; Data for Routine_0
DECL LDAT LCPDATP1={VEL 1,ACC 100,APO_DIST 5,APO_FAC 50.0,ORI_TYP #VAR,CIRC_TYP #BASE,JERK_FAC 50.0}
DECL FDAT FP1={TOOL_NO 2,BASE_NO 10,IPO_FRAME #BASE,POINT2[] " ",TQ_STATE FALSE}
DECL E6POS XP1={X -58.570,Y 107.870,Z -38.440,A 0.000,B -17.860,C -36.410}
DECL LDAT LCPDATC2={VEL 0.1,ACC 100,APO_DIST 5,APO_FAC 50.0,ORI_TYP #VAR,CIRC_TYP #BASE,JERK_FAC 50.0}
DECL FDAT FC2={TOOL_NO 2,BASE_NO 10,IPO_FRAME #BASE,POINT2[] " ",TQ_STATE FALSE}
DECL E6POS XCAux2={X -46.970,Y 113.400,Z -38.440,A 0.000,B -14.240,C -37.780}
DECL E6POS XCDes2={X 46.970,Y 113.400,Z -38.440,A 0.000,B 14.240,C -37.780}
DECL LDAT LCPDATP3={VEL 1,ACC 100,APO_DIST 5,APO_FAC 50.0,ORI_TYP #VAR,CIRC_TYP #BASE,JERK_FAC 50.0}
DECL FDAT FP3={TOOL_NO 2,BASE_NO 10,IPO_FRAME #BASE,POINT2[] " ",TQ_STATE FALSE}
DECL E6POS XP3={X 58.570,Y 107.870,Z -38.440,A 0.000,B 17.860,C -36.410}
DECL LDAT LCPDATP4={VEL 1,ACC 100,APO_DIST 5,APO_FAC 50.0,ORI_TYP #VAR,CIRC_TYP #BASE,JERK_FAC 50.0}
DECL FDAT FP4={TOOL_NO 2,BASE_NO 10,IPO_FRAME #BASE,POINT2[] " ",TQ_STATE FALSE}
DECL E6POS XP4={X 62.100,Y 114.380,Z -43.390,A 0.000,B 12.720,C -24.560}
DECL LDAT LCPDATC5={VEL 0.1,ACC 100,APO_DIST 5,APO_FAC 50.0,ORI_TYP #VAR,CIRC_TYP #BASE,JERK_FAC 50.0}
DECL FDAT FC5={TOOL_NO 2,BASE_NO 10,IPO_FRAME #BASE,POINT2[] " ",TQ_STATE FALSE}
DECL E6POS XCAux5={X 49.810,Y 120.250,Z -43.390,A 0.000,B 10.170,C -25.660}
DECL E6POS XCDes5={X -49.810,Y 120.250,Z -43.390,A -0.000,B -10.170,C -25.660}
DECL LDAT LCPDATP6={VEL 1,ACC 100,APO_DIST 5,APO_FAC 50.0,ORI_TYP #VAR,CIRC_TYP #BASE,JERK_FAC 50.0}
DECL FDAT FP6={TOOL_NO 2,BASE_NO 10,IPO_FRAME #BASE,POINT2[] " ",TQ_STATE FALSE}
DECL E6POS XP6={X -62.100,Y 114.380,Z -43.390,A 0.000,B -12.720,C -24.560}
DECL LDAT LCPDATP7={VEL 1,ACC 100,APO_DIST 5,APO_FAC 50.0,ORI_TYP #VAR,CIRC_TYP #BASE,JERK_FAC 50.0}
DECL FDAT FP7={TOOL_NO 2,BASE_NO 10,IPO_FRAME #BASE,POINT2[] " ",TQ_STATE FALSE}
DECL E6POS XP7={X -66.070,Y 121.680,Z -46.620,A -0.000,B -7.070,C -13.210}
DECL LDAT LCPDATC8={VEL 0.1,ACC 100,APO_DIST 5,APO_FAC 50.0,ORI_TYP #VAR,CIRC_TYP #BASE,JERK_FAC 50.0}
DECL FDAT FC8={TOOL_NO 2,BASE_NO 10,IPO_FRAME #BASE,POINT2[] " ",TQ_STATE FALSE}
DECL E6POS XCAux8={X -52.990,Y 127.920,Z -46.620,A 0.000,B -5.670,C -13.860}
DECL E6POS XCDes8={X 52.990,Y 127.920,Z -46.620,A 0.000,B 5.670,C -13.860}
DECL LDAT LCPDATP9={VEL 1,ACC 100,APO_DIST 5,APO_FAC 50.0,ORI_TYP #VAR,CIRC_TYP #BASE,JERK_FAC 50.0}
DECL FDAT FP9={TOOL_NO 2,BASE_NO 10,IPO_FRAME #BASE,POINT2[] " ",TQ_STATE FALSE}
DECL E6POS XP9={X 66.070,Y 121.680,Z -46.620,A 0.000,B 7.070,C -13.210}
DECL LDAT LCPDATP10={VEL 1,ACC 100,APO_DIST 5,APO_FAC 50.0,ORI_TYP #VAR,CIRC_TYP #BASE,JERK_FAC 50.0}
DECL FDAT FP10={TOOL_NO 2,BASE_NO 10,IPO_FRAME #BASE,POINT2[] " ",TQ_STATE FALSE}
DECL E6POS XP10={X 70.270,Y 129.420,Z -47.960,A 0.000,B 1.160,C -2.140}
DECL LDAT LCPDATC11={VEL 0.1,ACC 100,APO_DIST 5,APO_FAC 50.0,ORI_TYP #VAR,CIRC_TYP #BASE,JERK_FAC 50.0}
DECL FDAT FC11={TOOL_NO 2,BASE_NO 10,IPO_FRAME #BASE,POINT2[] " ",TQ_STATE FALSE}
DECL E6POS XCAux11={X 56.360,Y 136.060,Z -47.960,A 0.000,B 0.930,C -2.250}
DECL E6POS XCDes11={X -56.360,Y 136.060,Z -47.960,A 0.000,B -0.930,C -2.250}
DECL LDAT LCPDATP12={VEL 1,ACC 100,APO_DIST 5,APO_FAC 50.0,ORI_TYP #VAR,CIRC_TYP #BASE,JERK_FAC 50.0}
DECL FDAT FP12={TOOL_NO 2,BASE_NO 10,IPO_FRAME #BASE,POINT2[] " ",TQ_STATE FALSE}
DECL E6POS XP12={X -70.270,Y 129.420,Z -47.960,A 0.000,B -1.160,C -2.140}
DECL LDAT LCPDATP13={VEL 1,ACC 100,APO_DIST 5,APO_FAC 50.0,ORI_TYP #VAR,CIRC_TYP #BASE,JERK_FAC 50.0}
DECL FDAT FP13={TOOL_NO 2,BASE_NO 10,IPO_FRAME #BASE,POINT2[] " ",TQ_STATE FALSE}
DECL E6POS XP13={X -70.330,Y 129.530,Z -48.000,A 0.000,B 0.000,C -0.000}
DECL LDAT LCPDATC14={VEL 0.1,ACC 100,APO_DIST 5,APO_FAC 50.0,ORI_TYP #VAR,CIRC_TYP #BASE,JERK_FAC 50.0}
DECL FDAT FC14={TOOL_NO 2,BASE_NO 10,IPO_FRAME #BASE,POINT2[] " ",TQ_STATE FALSE}
DECL E6POS XCAux14={X -56.400,Y 136.170,Z -48.000,A 0.000,B 0.000,C -0.000}
DECL E6POS XCDes14={X 56.400,Y 136.170,Z -48.000,A 0.000,B 0.000,C -0.000}
DECL LDAT LCPDATP15={VEL 1,ACC 100,APO_DIST 5,APO_FAC 50.0,ORI_TYP #VAR,CIRC_TYP #BASE,JERK_FAC 50.0}
DECL FDAT FP15={TOOL_NO 2,BASE_NO 10,IPO_FRAME #BASE,POINT2[] " ",TQ_STATE FALSE}
DECL E6POS XP15={X 70.330,Y 129.530,Z -48.000,A 0.000,B 0.000,C -0.000}
DECL LDAT LCPDATP16={VEL 1,ACC 100,APO_DIST 5,APO_FAC 50.0,ORI_TYP #VAR,CIRC_TYP #BASE,JERK_FAC 50.0}
DECL FDAT FP16={TOOL_NO 2,BASE_NO 10,IPO_FRAME #BASE,POINT2[] " ",TQ_STATE FALSE}
DECL E6POS XP16={X 69.370,Y 127.770,Z -48.000,A 0.000,B 0.000,C -0.000}
DECL LDAT LCPDATC17={VEL 0.1,ACC 100,APO_DIST 5,APO_FAC 50.0,ORI_TYP #VAR,CIRC_TYP #BASE,JERK_FAC 50.0}
DECL FDAT FC17={TOOL_NO 2,BASE_NO 10,IPO_FRAME #BASE,POINT2[] " ",TQ_STATE FALSE}
DECL E6POS XCAux17={X 55.640,Y 134.320,Z -48.000,A 0.000,B 0.000,C -0.000}
DECL E6POS XCDes17={X -55.640,Y 134.320,Z -48.000,A 0.000,B 0.000,C -0.000}
DECL LDAT LCPDATP18={VEL 1,ACC 100,APO_DIST 5,APO_FAC 50.0,ORI_TYP #VAR,CIRC_TYP #BASE,JERK_FAC 50.0}
DECL FDAT FP18={TOOL_NO 2,BASE_NO 10,IPO_FRAME #BASE,POINT2[] " ",TQ_STATE FALSE}
DECL E6POS XP18={X -69.370,Y 127.770,Z -48.000,A 0.000,B 0.000,C -0.000}
DECL LDAT LCPDATP19={VEL 1,ACC 100,APO_DIST 5,APO_FAC 50.0,ORI_TYP #VAR,CIRC_TYP #BASE,JERK_FAC 50.0}
DECL FDAT FP19={TOOL_NO 2,BASE_NO 10,IPO_FRAME #BASE,POINT2[] " ",TQ_STATE FALSE}
DECL E6POS XP19={X -68.420,Y 126.010,Z -48.000,A 0.000,B 0.000,C -0.000}
DECL LDAT LCPDATC20={VEL 0.1,ACC 100,APO_DIST 5,APO_FAC 50.0,ORI_TYP #VAR,CIRC_TYP #BASE,JERK_FAC 50.0}
DECL FDAT FC20={TOOL_NO 2,BASE_NO 10,IPO_FRAME #BASE,POINT2[] " ",TQ_STATE FALSE}
DECL E6POS XCAux20={X -54.870,Y 132.470,Z -48.000,A 0.000,B 0.000,C -0.000}
DECL E6POS XCDes20={X 54.870,Y 132.470,Z -48.000,A 0.000,B 0.000,C -0.000}
DECL LDAT LCPDATP21={VEL 1,ACC 100,APO_DIST 5,APO_FAC 50.0,ORI_TYP #VAR,CIRC_TYP #BASE,JERK_FAC 50.0}
DECL FDAT FP21={TOOL_NO 2,BASE_NO 10,IPO_FRAME #BASE,POINT2[] " ",TQ_STATE FALSE}
DECL E6POS XP21={X 68.420,Y 126.010,Z -48.000,A 0.000,B 0.000,C -0.000}
DECL LDAT LCPDATP22={VEL 1,ACC 100,APO_DIST 5,APO_FAC 50.0,ORI_TYP #VAR,CIRC_TYP #BASE,JERK_FAC 50.0}
DECL FDAT FP22={TOOL_NO 2,BASE_NO 10,IPO_FRAME #BASE,POINT2[] " ",TQ_STATE FALSE}
DECL E6POS XP22={X 67.460,Y 124.250,Z -48.000,A 0.000,B 0.000,C -0.000}
DECL LDAT LCPDATC23={VEL 0.1,ACC 100,APO_DIST 5,APO_FAC 50.0,ORI_TYP #VAR,CIRC_TYP #BASE,JERK_FAC 50.0}
DECL FDAT FC23={TOOL_NO 2,BASE_NO 10,IPO_FRAME #BASE,POINT2[] " ",TQ_STATE FALSE}
DECL E6POS XCAux23={X 54.110,Y 130.630,Z -48.000,A 0.000,B 0.000,C -0.000}
DECL E6POS XCDes23={X -54.110,Y 130.630,Z -48.000,A 0.000,B 0.000,C -0.000}
DECL LDAT LCPDATP24={VEL 1,ACC 100,APO_DIST 5,APO_FAC 50.0,ORI_TYP #VAR,CIRC_TYP #BASE,JERK_FAC 50.0}
DECL FDAT FP24={TOOL_NO 2,BASE_NO 10,IPO_FRAME #BASE,POINT2[] " ",TQ_STATE FALSE}
DECL E6POS XP24={X -67.460,Y 124.250,Z -48.000,A 0.000,B 0.000,C -0.000}
DECL LDAT LCPDATP25={VEL 1,ACC 100,APO_DIST 5,APO_FAC 50.0,ORI_TYP #VAR,CIRC_TYP #BASE,JERK_FAC 50.0}
DECL FDAT FP25={TOOL_NO 2,BASE_NO 10,IPO_FRAME #BASE,POINT2[] " ",TQ_STATE FALSE}
DECL E6POS XP25={X -70.710,Y 130.240,Z -47.360,A 0.000,B 4.820,C 8.940}
DECL LDAT LCPDATC26={VEL 0.1,ACC 100,APO_DIST 5,APO_FAC 50.0,ORI_TYP #VAR,CIRC_TYP #BASE,JERK_FAC 50.0}
DECL FDAT FC26={TOOL_NO 2,BASE_NO 10,IPO_FRAME #BASE,POINT2[] " ",TQ_STATE FALSE}
DECL E6POS XCAux26={X -56.710,Y 136.910,Z -47.360,A 0.000,B 3.870,C 9.390}
DECL E6POS XCDes26={X 56.710,Y 136.910,Z -47.360,A 0.000,B -3.870,C 9.390}
DECL LDAT LCPDATP27={VEL 1,ACC 100,APO_DIST 5,APO_FAC 50.0,ORI_TYP #VAR,CIRC_TYP #BASE,JERK_FAC 50.0}
DECL FDAT FP27={TOOL_NO 2,BASE_NO 10,IPO_FRAME #BASE,POINT2[] " ",TQ_STATE FALSE}
DECL E6POS XP27={X 70.710,Y 130.240,Z -47.360,A -0.000,B -4.820,C 8.940}
DECL LDAT LCPDATP28={VEL 1,ACC 100,APO_DIST 5,APO_FAC 50.0,ORI_TYP #VAR,CIRC_TYP #BASE,JERK_FAC 50.0}
DECL FDAT FP28={TOOL_NO 2,BASE_NO 10,IPO_FRAME #BASE,POINT2[] " ",TQ_STATE FALSE}
DECL E6POS XP28={X 74.790,Y 137.750,Z -44.840,A -0.000,B -10.600,C 20.160}
DECL LDAT LCPDATC29={VEL 0.1,ACC 100,APO_DIST 5,APO_FAC 50.0,ORI_TYP #VAR,CIRC_TYP #BASE,JERK_FAC 50.0}
DECL FDAT FC29={TOOL_NO 2,BASE_NO 10,IPO_FRAME #BASE,POINT2[] " ",TQ_STATE FALSE}
DECL E6POS XCAux29={X 59.980,Y 144.810,Z -44.840,A -0.000,B -8.480,C 21.100}
DECL E6POS XCDes29={X -59.980,Y 144.810,Z -44.840,A -0.000,B 8.480,C 21.100}
DECL LDAT LCPDATP30={VEL 1,ACC 100,APO_DIST 5,APO_FAC 50.0,ORI_TYP #VAR,CIRC_TYP #BASE,JERK_FAC 50.0}
DECL FDAT FP30={TOOL_NO 2,BASE_NO 10,IPO_FRAME #BASE,POINT2[] " ",TQ_STATE FALSE}
DECL E6POS XP30={X -74.790,Y 137.750,Z -44.840,A 0.000,B 10.600,C 20.160}
DECL LDAT LCPDATP31={VEL 1,ACC 100,APO_DIST 5,APO_FAC 50.0,ORI_TYP #VAR,CIRC_TYP #BASE,JERK_FAC 50.0}
DECL FDAT FP31={TOOL_NO 2,BASE_NO 10,IPO_FRAME #BASE,POINT2[] " ",TQ_STATE FALSE}
DECL E6POS XP31={X -78.510,Y 144.600,Z -40.530,A 0.000,B 15.960,C 31.790}
DECL LDAT LCPDATC32={VEL 0.1,ACC 100,APO_DIST 5,APO_FAC 50.0,ORI_TYP #VAR,CIRC_TYP #BASE,JERK_FAC 50.0}
DECL FDAT FC32={TOOL_NO 2,BASE_NO 10,IPO_FRAME #BASE,POINT2[] " ",TQ_STATE FALSE}
DECL E6POS XCAux32={X -62.970,Y 152.020,Z -40.530,A 0.000,B 12.740,C 33.080}
DECL E6POS XCDes32={X 62.970,Y 152.020,Z -40.530,A 0.000,B -12.740,C 33.080}
DECL LDAT LCPDATP33={VEL 1,ACC 100,APO_DIST 5,APO_FAC 50.0,ORI_TYP #VAR,CIRC_TYP #BASE,JERK_FAC 50.0}
DECL FDAT FP33={TOOL_NO 2,BASE_NO 10,IPO_FRAME #BASE,POINT2[] " ",TQ_STATE FALSE}
DECL E6POS XP33={X 78.510,Y 144.600,Z -40.530,A 0.000,B -15.960,C 31.790}
DECL LDAT LCPDATP34={VEL 1,ACC 100,APO_DIST 5,APO_FAC 50.0,ORI_TYP #VAR,CIRC_TYP #BASE,JERK_FAC 50.0}
DECL FDAT FP34={TOOL_NO 2,BASE_NO 10,IPO_FRAME #BASE,POINT2[] " ",TQ_STATE FALSE}
DECL E6POS XP34={X 81.700,Y 150.470,Z -34.640,A 0.000,B -20.670,C 44.020}
DECL LDAT LCPDATC35={VEL 0.1,ACC 100,APO_DIST 5,APO_FAC 50.0,ORI_TYP #VAR,CIRC_TYP #BASE,JERK_FAC 50.0}
DECL FDAT FC35={TOOL_NO 2,BASE_NO 10,IPO_FRAME #BASE,POINT2[] " ",TQ_STATE FALSE}
DECL E6POS XCAux35={X 65.520,Y 158.190,Z -34.640,A 0.000,B -16.450,C 45.450}
DECL E6POS XCDes35={X -65.520,Y 158.190,Z -34.640,A 0.000,B 16.450,C 45.450}
DECL LDAT LCPDATP36={VEL 1,ACC 100,APO_DIST 5,APO_FAC 50.0,ORI_TYP #VAR,CIRC_TYP #BASE,JERK_FAC 50.0}
DECL FDAT FP36={TOOL_NO 2,BASE_NO 10,IPO_FRAME #BASE,POINT2[] " ",TQ_STATE FALSE}
DECL E6POS XP36={X -81.700,Y 150.470,Z -34.640,A 0.000,B 20.670,C 44.020}
DECL LDAT LCPDATP37={VEL 1,ACC 100,APO_DIST 5,APO_FAC 50.0,ORI_TYP #VAR,CIRC_TYP #BASE,JERK_FAC 50.0}
DECL FDAT FP37={TOOL_NO 2,BASE_NO 10,IPO_FRAME #BASE,POINT2[] " ",TQ_STATE FALSE}
DECL E6POS XP37={X -79.930,Y 147.210,Z -38.750,A -0.000,B 17.860,C 36.410}
DECL LDAT LCPDATC38={VEL 0.1,ACC 100,APO_DIST 5,APO_FAC 50.0,ORI_TYP #VAR,CIRC_TYP #BASE,JERK_FAC 50.0}
DECL FDAT FC38={TOOL_NO 2,BASE_NO 10,IPO_FRAME #BASE,POINT2[] " ",TQ_STATE FALSE}
DECL E6POS XCAux38={X -64.110,Y 154.760,Z -38.750,A -0.000,B 14.240,C 37.780}
DECL E6POS XCDes38={X 64.110,Y 154.760,Z -38.750,A 0.000,B -14.240,C 37.780}
DECL LDAT LCPDATP39={VEL 1,ACC 100,APO_DIST 5,APO_FAC 50.0,ORI_TYP #VAR,CIRC_TYP #BASE,JERK_FAC 50.0}
DECL FDAT FP39={TOOL_NO 2,BASE_NO 10,IPO_FRAME #BASE,POINT2[] " ",TQ_STATE FALSE}
DECL E6POS XP39={X 79.930,Y 147.210,Z -38.750,A -0.000,B -17.860,C 36.410}
DECL LDAT LCPDATP40={VEL 1,ACC 100,APO_DIST 5,APO_FAC 50.0,ORI_TYP #VAR,CIRC_TYP #BASE,JERK_FAC 50.0}
DECL FDAT FP40={TOOL_NO 2,BASE_NO 10,IPO_FRAME #BASE,POINT2[] " ",TQ_STATE FALSE}
DECL E6POS XP40={X 76.190,Y 140.320,Z -43.940,A -0.000,B -12.470,C 24.030}
DECL LDAT LCPDATC41={VEL 0.1,ACC 100,APO_DIST 5,APO_FAC 50.0,ORI_TYP #VAR,CIRC_TYP #BASE,JERK_FAC 50.0}
DECL FDAT FC41={TOOL_NO 2,BASE_NO 10,IPO_FRAME #BASE,POINT2[] " ",TQ_STATE FALSE}
DECL E6POS XCAux41={X 61.100,Y 147.510,Z -43.940,A -0.000,B -9.970,C 25.120}
DECL E6POS XCDes41={X -61.100,Y 147.510,Z -43.940,A 0.000,B 9.970,C 25.120}
DECL LDAT LCPDATP42={VEL 1,ACC 100,APO_DIST 5,APO_FAC 50.0,ORI_TYP #VAR,CIRC_TYP #BASE,JERK_FAC 50.0}
DECL FDAT FP42={TOOL_NO 2,BASE_NO 10,IPO_FRAME #BASE,POINT2[] " ",TQ_STATE FALSE}
DECL E6POS XP42={X -76.190,Y 140.320,Z -43.940,A 0.000,B 12.470,C 24.030}
DECL LDAT LCPDATP43={VEL 1,ACC 100,APO_DIST 5,APO_FAC 50.0,ORI_TYP #VAR,CIRC_TYP #BASE,JERK_FAC 50.0}
DECL FDAT FP43={TOOL_NO 2,BASE_NO 10,IPO_FRAME #BASE,POINT2[] " ",TQ_STATE FALSE}
DECL E6POS XP43={X -71.980,Y 132.570,Z -47.210,A 0.000,B 6.540,C 12.190}
DECL LDAT LCPDATC44={VEL 0.1,ACC 100,APO_DIST 5,APO_FAC 50.0,ORI_TYP #VAR,CIRC_TYP #BASE,JERK_FAC 50.0}
DECL FDAT FC44={TOOL_NO 2,BASE_NO 10,IPO_FRAME #BASE,POINT2[] " ",TQ_STATE FALSE}
DECL E6POS XCAux44={X -57.730,Y 139.360,Z -47.210,A 0.000,B 5.240,C 12.790}
DECL E6POS XCDes44={X 57.730,Y 139.360,Z -47.210,A 0.000,B -5.240,C 12.790}
DECL LDAT LCPDATP45={VEL 1,ACC 100,APO_DIST 5,APO_FAC 50.0,ORI_TYP #VAR,CIRC_TYP #BASE,JERK_FAC 50.0}
DECL FDAT FP45={TOOL_NO 2,BASE_NO 10,IPO_FRAME #BASE,POINT2[] " ",TQ_STATE FALSE}
DECL E6POS XP45={X 71.980,Y 132.570,Z -47.210,A 0.000,B -6.540,C 12.190}
DECL LDAT LCPDATP46={VEL 1,ACC 100,APO_DIST 5,APO_FAC 50.0,ORI_TYP #VAR,CIRC_TYP #BASE,JERK_FAC 50.0}
DECL FDAT FP46={TOOL_NO 2,BASE_NO 10,IPO_FRAME #BASE,POINT2[] " ",TQ_STATE FALSE}
DECL E6POS XP46={X 67.520,Y 124.360,Z -48.400,A 0.000,B -0.340,C 0.630}
DECL LDAT LCPDATC47={VEL 0.1,ACC 100,APO_DIST 5,APO_FAC 50.0,ORI_TYP #VAR,CIRC_TYP #BASE,JERK_FAC 50.0}
DECL FDAT FC47={TOOL_NO 2,BASE_NO 10,IPO_FRAME #BASE,POINT2[] " ",TQ_STATE FALSE}
DECL E6POS XCAux47={X 54.160,Y 130.740,Z -48.400,A -0.000,B -0.270,C 0.660}
DECL E6POS XCDes47={X -54.160,Y 130.740,Z -48.400,A 0.000,B 0.270,C 0.660}
DECL LDAT LCPDATP48={VEL 1,ACC 100,APO_DIST 5,APO_FAC 50.0,ORI_TYP #VAR,CIRC_TYP #BASE,JERK_FAC 50.0}
DECL FDAT FP48={TOOL_NO 2,BASE_NO 10,IPO_FRAME #BASE,POINT2[] " ",TQ_STATE FALSE}
DECL E6POS XP48={X -67.520,Y 124.360,Z -48.400,A 0.000,B 0.340,C 0.630}
DECL LDAT LCPDATP49={VEL 1,ACC 100,APO_DIST 5,APO_FAC 50.0,ORI_TYP #VAR,CIRC_TYP #BASE,JERK_FAC 50.0}
DECL FDAT FP49={TOOL_NO 2,BASE_NO 10,IPO_FRAME #BASE,POINT2[] " ",TQ_STATE FALSE}
DECL E6POS XP49={X -68.180,Y 125.580,Z -48.400,A 0.000,B 0.000,C -0.000}
DECL LDAT LCPDATC50={VEL 0.1,ACC 100,APO_DIST 5,APO_FAC 50.0,ORI_TYP #VAR,CIRC_TYP #BASE,JERK_FAC 50.0}
DECL FDAT FC50={TOOL_NO 2,BASE_NO 10,IPO_FRAME #BASE,POINT2[] " ",TQ_STATE FALSE}
DECL E6POS XCAux50={X -54.680,Y 132.010,Z -48.400,A 0.000,B 0.000,C -0.000}
DECL E6POS XCDes50={X 54.680,Y 132.010,Z -48.400,A 0.000,B 0.000,C -0.000}
DECL LDAT LCPDATP51={VEL 1,ACC 100,APO_DIST 5,APO_FAC 50.0,ORI_TYP #VAR,CIRC_TYP #BASE,JERK_FAC 50.0}
DECL FDAT FP51={TOOL_NO 2,BASE_NO 10,IPO_FRAME #BASE,POINT2[] " ",TQ_STATE FALSE}
DECL E6POS XP51={X 68.180,Y 125.580,Z -48.400,A 0.000,B 0.000,C -0.000}
DECL LDAT LCPDATP52={VEL 1,ACC 100,APO_DIST 5,APO_FAC 50.0,ORI_TYP #VAR,CIRC_TYP #BASE,JERK_FAC 50.0}
DECL FDAT FP52={TOOL_NO 2,BASE_NO 10,IPO_FRAME #BASE,POINT2[] " ",TQ_STATE FALSE}
DECL E6POS XP52={X 69.140,Y 127.330,Z -48.400,A 0.000,B 0.000,C -0.000}
DECL LDAT LCPDATC53={VEL 0.1,ACC 100,APO_DIST 5,APO_FAC 50.0,ORI_TYP #VAR,CIRC_TYP #BASE,JERK_FAC 50.0}
DECL FDAT FC53={TOOL_NO 2,BASE_NO 10,IPO_FRAME #BASE,POINT2[] " ",TQ_STATE FALSE}
DECL E6POS XCAux53={X 55.450,Y 133.860,Z -48.400,A 0.000,B 0.000,C -0.000}
DECL E6POS XCDes53={X -55.450,Y 133.860,Z -48.400,A 0.000,B 0.000,C -0.000}
DECL LDAT LCPDATP54={VEL 1,ACC 100,APO_DIST 5,APO_FAC 50.0,ORI_TYP #VAR,CIRC_TYP #BASE,JERK_FAC 50.0}
DECL FDAT FP54={TOOL_NO 2,BASE_NO 10,IPO_FRAME #BASE,POINT2[] " ",TQ_STATE FALSE}
DECL E6POS XP54={X -69.140,Y 127.330,Z -48.400,A 0.000,B 0.000,C -0.000}
DECL LDAT LCPDATP55={VEL 1,ACC 100,APO_DIST 5,APO_FAC 50.0,ORI_TYP #VAR,CIRC_TYP #BASE,JERK_FAC 50.0}
DECL FDAT FP55={TOOL_NO 2,BASE_NO 10,IPO_FRAME #BASE,POINT2[] " ",TQ_STATE FALSE}
DECL E6POS XP55={X -70.090,Y 129.090,Z -48.400,A 0.000,B 0.000,C -0.000}
DECL LDAT LCPDATC56={VEL 0.1,ACC 100,APO_DIST 5,APO_FAC 50.0,ORI_TYP #VAR,CIRC_TYP #BASE,JERK_FAC 50.0}
DECL FDAT FC56={TOOL_NO 2,BASE_NO 10,IPO_FRAME #BASE,POINT2[] " ",TQ_STATE FALSE}
DECL E6POS XCAux56={X -56.210,Y 135.710,Z -48.400,A 0.000,B 0.000,C -0.000}
DECL E6POS XCDes56={X 56.210,Y 135.710,Z -48.400,A 0.000,B 0.000,C -0.000}
DECL LDAT LCPDATP57={VEL 1,ACC 100,APO_DIST 5,APO_FAC 50.0,ORI_TYP #VAR,CIRC_TYP #BASE,JERK_FAC 50.0}
DECL FDAT FP57={TOOL_NO 2,BASE_NO 10,IPO_FRAME #BASE,POINT2[] " ",TQ_STATE FALSE}
DECL E6POS XP57={X 70.090,Y 129.090,Z -48.400,A 0.000,B 0.000,C -0.000}
DECL LDAT LCPDATP58={VEL 1,ACC 100,APO_DIST 5,APO_FAC 50.0,ORI_TYP #VAR,CIRC_TYP #BASE,JERK_FAC 50.0}
DECL FDAT FP58={TOOL_NO 2,BASE_NO 10,IPO_FRAME #BASE,POINT2[] " ",TQ_STATE FALSE}
DECL E6POS XP58={X 71.040,Y 130.850,Z -48.400,A 0.000,B 0.000,C -0.000}
DECL LDAT LCPDATC59={VEL 0.1,ACC 100,APO_DIST 5,APO_FAC 50.0,ORI_TYP #VAR,CIRC_TYP #BASE,JERK_FAC 50.0}
DECL FDAT FC59={TOOL_NO 2,BASE_NO 10,IPO_FRAME #BASE,POINT2[] " ",TQ_STATE FALSE}
DECL E6POS XCAux59={X 56.980,Y 137.560,Z -48.400,A 0.000,B 0.000,C -0.000}
DECL E6POS XCDes59={X -56.980,Y 137.560,Z -48.400,A 0.000,B 0.000,C -0.000}
DECL LDAT LCPDATP60={VEL 1,ACC 100,APO_DIST 5,APO_FAC 50.0,ORI_TYP #VAR,CIRC_TYP #BASE,JERK_FAC 50.0}
DECL FDAT FP60={TOOL_NO 2,BASE_NO 10,IPO_FRAME #BASE,POINT2[] " ",TQ_STATE FALSE}
DECL E6POS XP60={X -71.040,Y 130.850,Z -48.400,A 0.000,B 0.000,C -0.000}
DECL LDAT LCPDATP61={VEL 1,ACC 100,APO_DIST 5,APO_FAC 50.0,ORI_TYP #VAR,CIRC_TYP #BASE,JERK_FAC 50.0}
DECL FDAT FP61={TOOL_NO 2,BASE_NO 10,IPO_FRAME #BASE,POINT2[] " ",TQ_STATE FALSE}
DECL E6POS XP61={X -66.840,Y 123.110,Z -47.430,A 0.000,B -5.920,C -11.010}
DECL LDAT LCPDATC62={VEL 0.1,ACC 100,APO_DIST 5,APO_FAC 50.0,ORI_TYP #VAR,CIRC_TYP #BASE,JERK_FAC 50.0}
DECL FDAT FC62={TOOL_NO 2,BASE_NO 10,IPO_FRAME #BASE,POINT2[] " ",TQ_STATE FALSE}
DECL E6POS XCAux62={X -53.610,Y 129.420,Z -47.430,A 0.000,B -4.740,C -11.560}
DECL E6POS XCDes62={X 53.610,Y 129.420,Z -47.430,A 0.000,B 4.740,C -11.560}
DECL LDAT LCPDATP63={VEL 1,ACC 100,APO_DIST 5,APO_FAC 50.0,ORI_TYP #VAR,CIRC_TYP #BASE,JERK_FAC 50.0}
DECL FDAT FP63={TOOL_NO 2,BASE_NO 10,IPO_FRAME #BASE,POINT2[] " ",TQ_STATE FALSE}
DECL E6POS XP63={X 66.840,Y 123.110,Z -47.430,A 0.000,B 5.920,C -11.010}
DECL LDAT LCPDATP64={VEL 1,ACC 100,APO_DIST 5,APO_FAC 50.0,ORI_TYP #VAR,CIRC_TYP #BASE,JERK_FAC 50.0}
DECL FDAT FP64={TOOL_NO 2,BASE_NO 10,IPO_FRAME #BASE,POINT2[] " ",TQ_STATE FALSE}
DECL E6POS XP64={X 62.600,Y 115.290,Z -44.360,A 0.000,B 11.890,C -22.810}
DECL LDAT LCPDATC65={VEL 0.1,ACC 100,APO_DIST 5,APO_FAC 50.0,ORI_TYP #VAR,CIRC_TYP #BASE,JERK_FAC 50.0}
DECL FDAT FC65={TOOL_NO 2,BASE_NO 10,IPO_FRAME #BASE,POINT2[] " ",TQ_STATE FALSE}
DECL E6POS XCAux65={X 50.210,Y 121.210,Z -44.360,A 0.000,B 9.510,C -23.850}
DECL E6POS XCDes65={X -50.210,Y 121.210,Z -44.360,A 0.000,B -9.510,C -23.850}
DECL LDAT LCPDATP66={VEL 1,ACC 100,APO_DIST 5,APO_FAC 50.0,ORI_TYP #VAR,CIRC_TYP #BASE,JERK_FAC 50.0}
DECL FDAT FP66={TOOL_NO 2,BASE_NO 10,IPO_FRAME #BASE,POINT2[] " ",TQ_STATE FALSE}
DECL E6POS XP66={X -62.600,Y 115.290,Z -44.360,A 0.000,B -11.890,C -22.810}
DECL LDAT LCPDATP67={VEL 1,ACC 100,APO_DIST 5,APO_FAC 50.0,ORI_TYP #VAR,CIRC_TYP #BASE,JERK_FAC 50.0}
DECL FDAT FP67={TOOL_NO 2,BASE_NO 10,IPO_FRAME #BASE,POINT2[] " ",TQ_STATE FALSE}
DECL E6POS XP67={X -58.800,Y 108.290,Z -39.360,A -0.000,B -17.350,C -35.120}
DECL LDAT LCPDATC68={VEL 0.1,ACC 100,APO_DIST 5,APO_FAC 50.0,ORI_TYP #VAR,CIRC_TYP #BASE,JERK_FAC 50.0}
DECL FDAT FC68={TOOL_NO 2,BASE_NO 10,IPO_FRAME #BASE,POINT2[] " ",TQ_STATE FALSE}
DECL E6POS XCAux68={X -47.160,Y 113.850,Z -39.360,A 0.000,B -13.830,C -36.480}
DECL E6POS XCDes68={X 47.160,Y 113.850,Z -39.360,A 0.000,B 13.830,C -36.480}
DECL LDAT LCPDATP69={VEL 1,ACC 100,APO_DIST 5,APO_FAC 50.0,ORI_TYP #VAR,CIRC_TYP #BASE,JERK_FAC 50.0}
DECL FDAT FP69={TOOL_NO 2,BASE_NO 10,IPO_FRAME #BASE,POINT2[] " ",TQ_STATE FALSE}
DECL E6POS XP69={X 58.800,Y 108.290,Z -39.360,A 0.000,B 17.350,C -35.120}
DECL LDAT LCPDATP70={VEL 1,ACC 100,APO_DIST 5,APO_FAC 50.0,ORI_TYP #VAR,CIRC_TYP #BASE,JERK_FAC 50.0}
DECL FDAT FP70={TOOL_NO 2,BASE_NO 10,IPO_FRAME #BASE,POINT2[] " ",TQ_STATE FALSE}
DECL E6POS XP70={X 58.320,Y 107.420,Z -39.060,A -0.000,B 17.860,C -36.410}
DECL LDAT LCPDATC71={VEL 0.1,ACC 100,APO_DIST 5,APO_FAC 50.0,ORI_TYP #VAR,CIRC_TYP #BASE,JERK_FAC 50.0}
DECL FDAT FC71={TOOL_NO 2,BASE_NO 10,IPO_FRAME #BASE,POINT2[] " ",TQ_STATE FALSE}
DECL E6POS XCAux71={X 46.770,Y 112.920,Z -39.060,A 0.000,B 14.240,C -37.780}
DECL E6POS XCDes71={X -46.770,Y 112.920,Z -39.060,A -0.000,B -14.240,C -37.780}
DECL LDAT LCPDATP72={VEL 1,ACC 100,APO_DIST 5,APO_FAC 50.0,ORI_TYP #VAR,CIRC_TYP #BASE,JERK_FAC 50.0}
DECL FDAT FP72={TOOL_NO 2,BASE_NO 10,IPO_FRAME #BASE,POINT2[] " ",TQ_STATE FALSE}
DECL E6POS XP72={X -58.320,Y 107.420,Z -39.060,A -0.000,B -17.860,C -36.410}
DECL LDAT LCPDATP73={VEL 1,ACC 100,APO_DIST 5,APO_FAC 50.0,ORI_TYP #VAR,CIRC_TYP #BASE,JERK_FAC 50.0}
DECL FDAT FP73={TOOL_NO 2,BASE_NO 10,IPO_FRAME #BASE,POINT2[] " ",TQ_STATE FALSE}
DECL E6POS XP73={X -62.300,Y 114.740,Z -44.500,A 0.000,B -12.200,C -23.460}
DECL LDAT LCPDATC74={VEL 0.1,ACC 100,APO_DIST 5,APO_FAC 50.0,ORI_TYP #VAR,CIRC_TYP #BASE,JERK_FAC 50.0}
DECL FDAT FC74={TOOL_NO 2,BASE_NO 10,IPO_FRAME #BASE,POINT2[] " ",TQ_STATE FALSE}
DECL E6POS XCAux74={X -49.960,Y 120.620,Z -44.500,A -0.000,B -9.750,C -24.520}
DECL E6POS XCDes74={X 49.960,Y 120.620,Z -44.500,A -0.000,B 9.750,C -24.520}
DECL LDAT LCPDATP75={VEL 1,ACC 100,APO_DIST 5,APO_FAC 50.0,ORI_TYP #VAR,CIRC_TYP #BASE,JERK_FAC 50.0}
DECL FDAT FP75={TOOL_NO 2,BASE_NO 10,IPO_FRAME #BASE,POINT2[] " ",TQ_STATE FALSE}
DECL E6POS XP75={X 62.300,Y 114.740,Z -44.500,A -0.000,B 12.200,C -23.460}
DECL LDAT LCPDATP76={VEL 1,ACC 100,APO_DIST 5,APO_FAC 50.0,ORI_TYP #VAR,CIRC_TYP #BASE,JERK_FAC 50.0}
DECL FDAT FP76={TOOL_NO 2,BASE_NO 10,IPO_FRAME #BASE,POINT2[] " ",TQ_STATE FALSE}
DECL E6POS XP76={X 66.780,Y 122.990,Z -47.800,A 0.000,B 5.950,C -11.070}
DECL LDAT LCPDATC77={VEL 0.1,ACC 100,APO_DIST 5,APO_FAC 50.0,ORI_TYP #VAR,CIRC_TYP #BASE,JERK_FAC 50.0}
DECL FDAT FC77={TOOL_NO 2,BASE_NO 10,IPO_FRAME #BASE,POINT2[] " ",TQ_STATE FALSE}
DECL E6POS XCAux77={X 53.560,Y 129.290,Z -47.800,A 0.000,B 4.770,C -11.630}
DECL E6POS XCDes77={X -53.560,Y 129.290,Z -47.800,A 0.000,B -4.770,C -11.630}
DECL LDAT LCPDATP78={VEL 1,ACC 100,APO_DIST 5,APO_FAC 50.0,ORI_TYP #VAR,CIRC_TYP #BASE,JERK_FAC 50.0}
DECL FDAT FP78={TOOL_NO 2,BASE_NO 10,IPO_FRAME #BASE,POINT2[] " ",TQ_STATE FALSE}
DECL E6POS XP78={X -66.780,Y 122.990,Z -47.800,A 0.000,B -5.950,C -11.070}
DECL LDAT LCPDATP79={VEL 1,ACC 100,APO_DIST 5,APO_FAC 50.0,ORI_TYP #VAR,CIRC_TYP #BASE,JERK_FAC 50.0}
DECL FDAT FP79={TOOL_NO 2,BASE_NO 10,IPO_FRAME #BASE,POINT2[] " ",TQ_STATE FALSE}
DECL E6POS XP79={X -71.010,Y 130.780,Z -48.800,A 0.000,B 0.000,C -0.000}
DECL LDAT LCPDATC80={VEL 0.1,ACC 100,APO_DIST 5,APO_FAC 50.0,ORI_TYP #VAR,CIRC_TYP #BASE,JERK_FAC 50.0}
DECL FDAT FC80={TOOL_NO 2,BASE_NO 10,IPO_FRAME #BASE,POINT2[] " ",TQ_STATE FALSE}
DECL E6POS XCAux80={X -56.950,Y 137.490,Z -48.800,A 0.000,B 0.000,C -0.000}
DECL E6POS XCDes80={X 56.950,Y 137.490,Z -48.800,A 0.000,B 0.000,C -0.000}
DECL LDAT LCPDATP81={VEL 1,ACC 100,APO_DIST 5,APO_FAC 50.0,ORI_TYP #VAR,CIRC_TYP #BASE,JERK_FAC 50.0}
DECL FDAT FP81={TOOL_NO 2,BASE_NO 10,IPO_FRAME #BASE,POINT2[] " ",TQ_STATE FALSE}
DECL E6POS XP81={X 71.010,Y 130.780,Z -48.800,A 0.000,B 0.000,C -0.000}
DECL LDAT LCPDATP82={VEL 1,ACC 100,APO_DIST 5,APO_FAC 50.0,ORI_TYP #VAR,CIRC_TYP #BASE,JERK_FAC 50.0}
DECL FDAT FP82={TOOL_NO 2,BASE_NO 10,IPO_FRAME #BASE,POINT2[] " ",TQ_STATE FALSE}
DECL E6POS XP82={X 70.050,Y 129.020,Z -48.800,A 0.000,B 0.000,C -0.000}
DECL LDAT LCPDATC83={VEL 0.1,ACC 100,APO_DIST 5,APO_FAC 50.0,ORI_TYP #VAR,CIRC_TYP #BASE,JERK_FAC 50.0}
DECL FDAT FC83={TOOL_NO 2,BASE_NO 10,IPO_FRAME #BASE,POINT2[] " ",TQ_STATE FALSE}
DECL E6POS XCAux83={X 56.180,Y 135.640,Z -48.800,A 0.000,B 0.000,C -0.000}
DECL E6POS XCDes83={X -56.180,Y 135.640,Z -48.800,A 0.000,B 0.000,C -0.000}
DECL LDAT LCPDATP84={VEL 1,ACC 100,APO_DIST 5,APO_FAC 50.0,ORI_TYP #VAR,CIRC_TYP #BASE,JERK_FAC 50.0}
DECL FDAT FP84={TOOL_NO 2,BASE_NO 10,IPO_FRAME #BASE,POINT2[] " ",TQ_STATE FALSE}
DECL E6POS XP84={X -70.050,Y 129.020,Z -48.800,A 0.000,B 0.000,C -0.000}
DECL LDAT LCPDATP85={VEL 1,ACC 100,APO_DIST 5,APO_FAC 50.0,ORI_TYP #VAR,CIRC_TYP #BASE,JERK_FAC 50.0}
DECL FDAT FP85={TOOL_NO 2,BASE_NO 10,IPO_FRAME #BASE,POINT2[] " ",TQ_STATE FALSE}
DECL E6POS XP85={X -69.100,Y 127.270,Z -48.800,A 0.000,B 0.000,C -0.000}
DECL LDAT LCPDATC86={VEL 0.1,ACC 100,APO_DIST 5,APO_FAC 50.0,ORI_TYP #VAR,CIRC_TYP #BASE,JERK_FAC 50.0}
DECL FDAT FC86={TOOL_NO 2,BASE_NO 10,IPO_FRAME #BASE,POINT2[] " ",TQ_STATE FALSE}
DECL E6POS XCAux86={X -55.420,Y 133.790,Z -48.800,A 0.000,B 0.000,C -0.000}
DECL E6POS XCDes86={X 55.420,Y 133.790,Z -48.800,A 0.000,B 0.000,C -0.000}
DECL LDAT LCPDATP87={VEL 1,ACC 100,APO_DIST 5,APO_FAC 50.0,ORI_TYP #VAR,CIRC_TYP #BASE,JERK_FAC 50.0}
DECL FDAT FP87={TOOL_NO 2,BASE_NO 10,IPO_FRAME #BASE,POINT2[] " ",TQ_STATE FALSE}
DECL E6POS XP87={X 69.100,Y 127.270,Z -48.800,A 0.000,B 0.000,C -0.000}
DECL LDAT LCPDATP88={VEL 1,ACC 100,APO_DIST 5,APO_FAC 50.0,ORI_TYP #VAR,CIRC_TYP #BASE,JERK_FAC 50.0}
DECL FDAT FP88={TOOL_NO 2,BASE_NO 10,IPO_FRAME #BASE,POINT2[] " ",TQ_STATE FALSE}
DECL E6POS XP88={X 68.150,Y 125.510,Z -48.800,A 0.000,B 0.000,C -0.000}
DECL LDAT LCPDATC89={VEL 0.1,ACC 100,APO_DIST 5,APO_FAC 50.0,ORI_TYP #VAR,CIRC_TYP #BASE,JERK_FAC 50.0}
DECL FDAT FC89={TOOL_NO 2,BASE_NO 10,IPO_FRAME #BASE,POINT2[] " ",TQ_STATE FALSE}
DECL E6POS XCAux89={X 54.650,Y 131.940,Z -48.800,A 0.000,B 0.000,C -0.000}
DECL E6POS XCDes89={X -54.650,Y 131.940,Z -48.800,A 0.000,B 0.000,C -0.000}
DECL LDAT LCPDATP90={VEL 1,ACC 100,APO_DIST 5,APO_FAC 50.0,ORI_TYP #VAR,CIRC_TYP #BASE,JERK_FAC 50.0}
DECL FDAT FP90={TOOL_NO 2,BASE_NO 10,IPO_FRAME #BASE,POINT2[] " ",TQ_STATE FALSE}
DECL E6POS XP90={X -68.150,Y 125.510,Z -48.800,A 0.000,B 0.000,C -0.000}
DECL LDAT LCPDATP91={VEL 1,ACC 100,APO_DIST 5,APO_FAC 50.0,ORI_TYP #VAR,CIRC_TYP #BASE,JERK_FAC 50.0}
DECL FDAT FP91={TOOL_NO 2,BASE_NO 10,IPO_FRAME #BASE,POINT2[] " ",TQ_STATE FALSE}
DECL E6POS XP91={X -67.720,Y 124.720,Z -48.790,A -0.000,B 0.610,C 1.110}
DECL LDAT LCPDATC92={VEL 0.1,ACC 100,APO_DIST 5,APO_FAC 50.0,ORI_TYP #VAR,CIRC_TYP #BASE,JERK_FAC 50.0}
DECL FDAT FC92={TOOL_NO 2,BASE_NO 10,IPO_FRAME #BASE,POINT2[] " ",TQ_STATE FALSE}
DECL E6POS XCAux92={X -54.310,Y 131.120,Z -48.790,A 0.000,B 0.490,C 1.170}
DECL E6POS XCDes92={X 54.310,Y 131.120,Z -48.790,A -0.000,B -0.490,C 1.170}
DECL LDAT LCPDATP93={VEL 1,ACC 100,APO_DIST 5,APO_FAC 50.0,ORI_TYP #VAR,CIRC_TYP #BASE,JERK_FAC 50.0}
DECL FDAT FP93={TOOL_NO 2,BASE_NO 10,IPO_FRAME #BASE,POINT2[] " ",TQ_STATE FALSE}
DECL E6POS XP93={X 67.720,Y 124.720,Z -48.790,A 0.000,B -0.610,C 1.110}
DECL LDAT LCPDATP94={VEL 1,ACC 100,APO_DIST 5,APO_FAC 50.0,ORI_TYP #VAR,CIRC_TYP #BASE,JERK_FAC 50.0}
DECL FDAT FP94={TOOL_NO 2,BASE_NO 10,IPO_FRAME #BASE,POINT2[] " ",TQ_STATE FALSE}
DECL E6POS XP94={X 72.420,Y 133.380,Z -47.380,A 0.000,B -7.090,C 13.240}
DECL LDAT LCPDATC95={VEL 0.1,ACC 100,APO_DIST 5,APO_FAC 50.0,ORI_TYP #VAR,CIRC_TYP #BASE,JERK_FAC 50.0}
DECL FDAT FC95={TOOL_NO 2,BASE_NO 10,IPO_FRAME #BASE,POINT2[] " ",TQ_STATE FALSE}
DECL E6POS XCAux95={X 58.080,Y 140.220,Z -47.380,A -0.000,B -5.680,C 13.900}
DECL E6POS XCDes95={X -58.080,Y 140.220,Z -47.380,A -0.000,B 5.680,C 13.900}
DECL LDAT LCPDATP96={VEL 1,ACC 100,APO_DIST 5,APO_FAC 50.0,ORI_TYP #VAR,CIRC_TYP #BASE,JERK_FAC 50.0}
DECL FDAT FP96={TOOL_NO 2,BASE_NO 10,IPO_FRAME #BASE,POINT2[] " ",TQ_STATE FALSE}
DECL E6POS XP96={X -72.420,Y 133.380,Z -47.380,A 0.000,B 7.090,C 13.240}
DECL LDAT LCPDATP97={VEL 1,ACC 100,APO_DIST 5,APO_FAC 50.0,ORI_TYP #VAR,CIRC_TYP #BASE,JERK_FAC 50.0}
DECL FDAT FP97={TOOL_NO 2,BASE_NO 10,IPO_FRAME #BASE,POINT2[] " ",TQ_STATE FALSE}
DECL E6POS XP97={X -76.830,Y 141.500,Z -43.680,A -0.000,B 13.250,C 25.710}
DECL LDAT LCPDATC98={VEL 0.1,ACC 100,APO_DIST 5,APO_FAC 50.0,ORI_TYP #VAR,CIRC_TYP #BASE,JERK_FAC 50.0}
DECL FDAT FC98={TOOL_NO 2,BASE_NO 10,IPO_FRAME #BASE,POINT2[] " ",TQ_STATE FALSE}
DECL E6POS XCAux98={X -61.620,Y 148.750,Z -43.680,A 0.000,B 10.590,C 26.840}
DECL E6POS XCDes98={X 61.620,Y 148.750,Z -43.680,A 0.000,B -10.590,C 26.840}
DECL LDAT LCPDATP99={VEL 1,ACC 100,APO_DIST 5,APO_FAC 50.0,ORI_TYP #VAR,CIRC_TYP #BASE,JERK_FAC 50.0}
DECL FDAT FP99={TOOL_NO 2,BASE_NO 10,IPO_FRAME #BASE,POINT2[] " ",TQ_STATE FALSE}
DECL E6POS XP99={X 76.830,Y 141.500,Z -43.680,A -0.000,B -13.250,C 25.710}
DECL LDAT LCPDATP100={VEL 1,ACC 100,APO_DIST 5,APO_FAC 50.0,ORI_TYP #VAR,CIRC_TYP #BASE,JERK_FAC 50.0}
DECL FDAT FP100={TOOL_NO 2,BASE_NO 10,IPO_FRAME #BASE,POINT2[] " ",TQ_STATE FALSE}
DECL E6POS XP100={X 80.690,Y 148.610,Z -37.890,A 0.000,B -18.780,C 38.780}
DECL LDAT LCPDATC101={VEL 0.1,ACC 100,APO_DIST 5,APO_FAC 50.0,ORI_TYP #VAR,CIRC_TYP #BASE,JERK_FAC 50.0}
DECL FDAT FC101={TOOL_NO 2,BASE_NO 10,IPO_FRAME #BASE,POINT2[] " ",TQ_STATE FALSE}
DECL E6POS XCAux101={X 64.710,Y 156.230,Z -37.890,A 0.000,B -14.960,C 40.190}
DECL E6POS XCDes101={X -64.710,Y 156.230,Z -37.890,A -0.000,B 14.960,C 40.190}
DECL LDAT LCPDATP102={VEL 1,ACC 100,APO_DIST 5,APO_FAC 50.0,ORI_TYP #VAR,CIRC_TYP #BASE,JERK_FAC 50.0}
DECL FDAT FP102={TOOL_NO 2,BASE_NO 10,IPO_FRAME #BASE,POINT2[] " ",TQ_STATE FALSE}
DECL E6POS XP102={X -80.690,Y 148.610,Z -37.890,A -0.000,B 18.780,C 38.780}
DECL LDAT LCPDATP103={VEL 1,ACC 100,APO_DIST 5,APO_FAC 50.0,ORI_TYP #VAR,CIRC_TYP #BASE,JERK_FAC 50.0}
DECL FDAT FP103={TOOL_NO 2,BASE_NO 10,IPO_FRAME #BASE,POINT2[] " ",TQ_STATE FALSE}
DECL E6POS XP103={X -80.180,Y 147.670,Z -39.360,A -0.000,B 17.860,C 36.410}
DECL LDAT LCPDATC104={VEL 0.1,ACC 100,APO_DIST 5,APO_FAC 50.0,ORI_TYP #VAR,CIRC_TYP #BASE,JERK_FAC 50.0}
DECL FDAT FC104={TOOL_NO 2,BASE_NO 10,IPO_FRAME #BASE,POINT2[] " ",TQ_STATE FALSE}
DECL E6POS XCAux104={X -64.300,Y 155.240,Z -39.360,A -0.000,B 14.240,C 37.780}
DECL E6POS XCDes104={X 64.300,Y 155.240,Z -39.360,A 0.000,B -14.240,C 37.780}
DECL LDAT LCPDATP105={VEL 1,ACC 100,APO_DIST 5,APO_FAC 50.0,ORI_TYP #VAR,CIRC_TYP #BASE,JERK_FAC 50.0}
DECL FDAT FP105={TOOL_NO 2,BASE_NO 10,IPO_FRAME #BASE,POINT2[] " ",TQ_STATE FALSE}
DECL E6POS XP105={X 80.180,Y 147.670,Z -39.360,A -0.000,B -17.860,C 36.410}
DECL LDAT LCPDATP106={VEL 1,ACC 100,APO_DIST 5,APO_FAC 50.0,ORI_TYP #VAR,CIRC_TYP #BASE,JERK_FAC 50.0}
DECL FDAT FP106={TOOL_NO 2,BASE_NO 10,IPO_FRAME #BASE,POINT2[] " ",TQ_STATE FALSE}
DECL E6POS XP106={X 75.940,Y 139.870,Z -45.080,A 0.000,B -11.890,C 22.820}
DECL LDAT LCPDATC107={VEL 0.1,ACC 100,APO_DIST 5,APO_FAC 50.0,ORI_TYP #VAR,CIRC_TYP #BASE,JERK_FAC 50.0}
DECL FDAT FC107={TOOL_NO 2,BASE_NO 10,IPO_FRAME #BASE,POINT2[] " ",TQ_STATE FALSE}
DECL E6POS XCAux107={X 60.910,Y 147.040,Z -45.080,A -0.000,B -9.510,C 23.860}
DECL E6POS XCDes107={X -60.910,Y 147.040,Z -45.080,A -0.000,B 9.510,C 23.860}
DECL LDAT LCPDATP108={VEL 1,ACC 100,APO_DIST 5,APO_FAC 50.0,ORI_TYP #VAR,CIRC_TYP #BASE,JERK_FAC 50.0}
DECL FDAT FP108={TOOL_NO 2,BASE_NO 10,IPO_FRAME #BASE,POINT2[] " ",TQ_STATE FALSE}
DECL E6POS XP108={X -75.940,Y 139.870,Z -45.080,A -0.000,B 11.890,C 22.820}
DECL LDAT LCPDATP109={VEL 1,ACC 100,APO_DIST 5,APO_FAC 50.0,ORI_TYP #VAR,CIRC_TYP #BASE,JERK_FAC 50.0}
DECL FDAT FP109={TOOL_NO 2,BASE_NO 10,IPO_FRAME #BASE,POINT2[] " ",TQ_STATE FALSE}
DECL E6POS XP109={X -71.170,Y 131.070,Z -48.400,A -0.000,B 5.310,C 9.850}
DECL LDAT LCPDATC110={VEL 0.1,ACC 100,APO_DIST 5,APO_FAC 50.0,ORI_TYP #VAR,CIRC_TYP #BASE,JERK_FAC 50.0}
DECL FDAT FC110={TOOL_NO 2,BASE_NO 10,IPO_FRAME #BASE,POINT2[] " ",TQ_STATE FALSE}
DECL E6POS XCAux110={X -57.080,Y 137.800,Z -48.400,A -0.000,B 4.250,C 10.340}
DECL E6POS XCDes110={X 57.080,Y 137.800,Z -48.400,A 0.000,B -4.250,C 10.340}
DECL LDAT LCPDATP111={VEL 1,ACC 100,APO_DIST 5,APO_FAC 50.0,ORI_TYP #VAR,CIRC_TYP #BASE,JERK_FAC 50.0}
DECL FDAT FP111={TOOL_NO 2,BASE_NO 10,IPO_FRAME #BASE,POINT2[] " ",TQ_STATE FALSE}
DECL E6POS XP111={X 71.170,Y 131.070,Z -48.400,A 0.000,B -5.310,C 9.850}
DECL LDAT LCPDATP112={VEL 1,ACC 100,APO_DIST 5,APO_FAC 50.0,ORI_TYP #VAR,CIRC_TYP #BASE,JERK_FAC 50.0}
DECL FDAT FP112={TOOL_NO 2,BASE_NO 10,IPO_FRAME #BASE,POINT2[] " ",TQ_STATE FALSE}
DECL E6POS XP112={X 67.500,Y 124.320,Z -49.200,A 0.000,B 0.000,C -0.000}
DECL LDAT LCPDATC113={VEL 0.1,ACC 100,APO_DIST 5,APO_FAC 50.0,ORI_TYP #VAR,CIRC_TYP #BASE,JERK_FAC 50.0}
DECL FDAT FC113={TOOL_NO 2,BASE_NO 10,IPO_FRAME #BASE,POINT2[] " ",TQ_STATE FALSE}
DECL E6POS XCAux113={X 54.130,Y 130.690,Z -49.200,A 0.000,B 0.000,C -0.000}
DECL E6POS XCDes113={X -54.130,Y 130.690,Z -49.200,A 0.000,B 0.000,C -0.000}
DECL LDAT LCPDATP114={VEL 1,ACC 100,APO_DIST 5,APO_FAC 50.0,ORI_TYP #VAR,CIRC_TYP #BASE,JERK_FAC 50.0}
DECL FDAT FP114={TOOL_NO 2,BASE_NO 10,IPO_FRAME #BASE,POINT2[] " ",TQ_STATE FALSE}
DECL E6POS XP114={X -67.500,Y 124.320,Z -49.200,A 0.000,B 0.000,C -0.000}
DECL LDAT LCPDATP115={VEL 1,ACC 100,APO_DIST 5,APO_FAC 50.0,ORI_TYP #VAR,CIRC_TYP #BASE,JERK_FAC 50.0}
DECL FDAT FP115={TOOL_NO 2,BASE_NO 10,IPO_FRAME #BASE,POINT2[] " ",TQ_STATE FALSE}
DECL E6POS XP115={X -68.450,Y 126.070,Z -49.200,A 0.000,B 0.000,C -0.000}
DECL LDAT LCPDATC116={VEL 0.1,ACC 100,APO_DIST 5,APO_FAC 50.0,ORI_TYP #VAR,CIRC_TYP #BASE,JERK_FAC 50.0}
DECL FDAT FC116={TOOL_NO 2,BASE_NO 10,IPO_FRAME #BASE,POINT2[] " ",TQ_STATE FALSE}
DECL E6POS XCAux116={X -54.900,Y 132.540,Z -49.200,A 0.000,B 0.000,C -0.000}
DECL E6POS XCDes116={X 54.900,Y 132.540,Z -49.200,A 0.000,B 0.000,C -0.000}
DECL LDAT LCPDATP117={VEL 1,ACC 100,APO_DIST 5,APO_FAC 50.0,ORI_TYP #VAR,CIRC_TYP #BASE,JERK_FAC 50.0}
DECL FDAT FP117={TOOL_NO 2,BASE_NO 10,IPO_FRAME #BASE,POINT2[] " ",TQ_STATE FALSE}
DECL E6POS XP117={X 68.450,Y 126.070,Z -49.200,A 0.000,B 0.000,C -0.000}
DECL LDAT LCPDATP118={VEL 1,ACC 100,APO_DIST 5,APO_FAC 50.0,ORI_TYP #VAR,CIRC_TYP #BASE,JERK_FAC 50.0}
DECL FDAT FP118={TOOL_NO 2,BASE_NO 10,IPO_FRAME #BASE,POINT2[] " ",TQ_STATE FALSE}
DECL E6POS XP118={X 69.410,Y 127.830,Z -49.200,A 0.000,B 0.000,C -0.000}
DECL LDAT LCPDATC119={VEL 0.1,ACC 100,APO_DIST 5,APO_FAC 50.0,ORI_TYP #VAR,CIRC_TYP #BASE,JERK_FAC 50.0}
DECL FDAT FC119={TOOL_NO 2,BASE_NO 10,IPO_FRAME #BASE,POINT2[] " ",TQ_STATE FALSE}
DECL E6POS XCAux119={X 55.660,Y 134.390,Z -49.200,A 0.000,B 0.000,C -0.000}
DECL E6POS XCDes119={X -55.660,Y 134.390,Z -49.200,A 0.000,B 0.000,C -0.000}
DECL LDAT LCPDATP120={VEL 1,ACC 100,APO_DIST 5,APO_FAC 50.0,ORI_TYP #VAR,CIRC_TYP #BASE,JERK_FAC 50.0}
DECL FDAT FP120={TOOL_NO 2,BASE_NO 10,IPO_FRAME #BASE,POINT2[] " ",TQ_STATE FALSE}
DECL E6POS XP120={X -69.410,Y 127.830,Z -49.200,A 0.000,B 0.000,C -0.000}
DECL LDAT LCPDATP121={VEL 1,ACC 100,APO_DIST 5,APO_FAC 50.0,ORI_TYP #VAR,CIRC_TYP #BASE,JERK_FAC 50.0}
DECL FDAT FP121={TOOL_NO 2,BASE_NO 10,IPO_FRAME #BASE,POINT2[] " ",TQ_STATE FALSE}
DECL E6POS XP121={X -70.360,Y 129.590,Z -49.200,A 0.000,B 0.000,C -0.000}
DECL LDAT LCPDATC122={VEL 0.1,ACC 100,APO_DIST 5,APO_FAC 50.0,ORI_TYP #VAR,CIRC_TYP #BASE,JERK_FAC 50.0}
DECL FDAT FC122={TOOL_NO 2,BASE_NO 10,IPO_FRAME #BASE,POINT2[] " ",TQ_STATE FALSE}
DECL E6POS XCAux122={X -56.430,Y 136.230,Z -49.200,A 0.000,B 0.000,C -0.000}
DECL E6POS XCDes122={X 56.430,Y 136.230,Z -49.200,A 0.000,B 0.000,C -0.000}
DECL LDAT LCPDATP123={VEL 1,ACC 100,APO_DIST 5,APO_FAC 50.0,ORI_TYP #VAR,CIRC_TYP #BASE,JERK_FAC 50.0}
DECL FDAT FP123={TOOL_NO 2,BASE_NO 10,IPO_FRAME #BASE,POINT2[] " ",TQ_STATE FALSE}
DECL E6POS XP123={X 70.360,Y 129.590,Z -49.200,A 0.000,B 0.000,C -0.000}
DECL LDAT LCPDATP124={VEL 1,ACC 100,APO_DIST 5,APO_FAC 50.0,ORI_TYP #VAR,CIRC_TYP #BASE,JERK_FAC 50.0}
DECL FDAT FP124={TOOL_NO 2,BASE_NO 10,IPO_FRAME #BASE,POINT2[] " ",TQ_STATE FALSE}
DECL E6POS XP124={X 69.940,Y 128.810,Z -49.130,A 0.000,B 1.580,C -2.910}
DECL LDAT LCPDATC125={VEL 0.1,ACC 100,APO_DIST 5,APO_FAC 50.0,ORI_TYP #VAR,CIRC_TYP #BASE,JERK_FAC 50.0}
DECL FDAT FC125={TOOL_NO 2,BASE_NO 10,IPO_FRAME #BASE,POINT2[] " ",TQ_STATE FALSE}
DECL E6POS XCAux125={X 56.090,Y 135.410,Z -49.130,A -0.000,B 1.270,C -3.060}
DECL E6POS XCDes125={X -56.090,Y 135.410,Z -49.130,A 0.000,B -1.270,C -3.060}
DECL LDAT LCPDATP126={VEL 1,ACC 100,APO_DIST 5,APO_FAC 50.0,ORI_TYP #VAR,CIRC_TYP #BASE,JERK_FAC 50.0}
DECL FDAT FP126={TOOL_NO 2,BASE_NO 10,IPO_FRAME #BASE,POINT2[] " ",TQ_STATE FALSE}
DECL E6POS XP126={X -69.940,Y 128.810,Z -49.130,A 0.000,B -1.580,C -2.910}
DECL LDAT LCPDATP127={VEL 1,ACC 100,APO_DIST 5,APO_FAC 50.0,ORI_TYP #VAR,CIRC_TYP #BASE,JERK_FAC 50.0}
DECL FDAT FP127={TOOL_NO 2,BASE_NO 10,IPO_FRAME #BASE,POINT2[] " ",TQ_STATE FALSE}
DECL E6POS XP127={X -64.990,Y 119.690,Z -47.200,A 0.000,B -8.350,C -15.690}
DECL LDAT LCPDATC128={VEL 0.1,ACC 100,APO_DIST 5,APO_FAC 50.0,ORI_TYP #VAR,CIRC_TYP #BASE,JERK_FAC 50.0}
DECL FDAT FC128={TOOL_NO 2,BASE_NO 10,IPO_FRAME #BASE,POINT2[] " ",TQ_STATE FALSE}
DECL E6POS XCAux128={X -52.120,Y 125.830,Z -47.200,A 0.000,B -6.690,C -16.450}
DECL E6POS XCDes128={X 52.120,Y 125.830,Z -47.200,A 0.000,B 6.690,C -16.450}
DECL LDAT LCPDATP129={VEL 1,ACC 100,APO_DIST 5,APO_FAC 50.0,ORI_TYP #VAR,CIRC_TYP #BASE,JERK_FAC 50.0}
DECL FDAT FP129={TOOL_NO 2,BASE_NO 10,IPO_FRAME #BASE,POINT2[] " ",TQ_STATE FALSE}
DECL E6POS XP129={X 64.990,Y 119.690,Z -47.200,A -0.000,B 8.350,C -15.690}
DECL LDAT LCPDATP130={VEL 1,ACC 100,APO_DIST 5,APO_FAC 50.0,ORI_TYP #VAR,CIRC_TYP #BASE,JERK_FAC 50.0}
DECL FDAT FP130={TOOL_NO 2,BASE_NO 10,IPO_FRAME #BASE,POINT2[] " ",TQ_STATE FALSE}
DECL E6POS XP130={X 60.420,Y 111.290,Z -42.760,A -0.000,B 14.700,C -28.900}
DECL LDAT LCPDATC131={VEL 0.1,ACC 100,APO_DIST 5,APO_FAC 50.0,ORI_TYP #VAR,CIRC_TYP #BASE,JERK_FAC 50.0}
DECL FDAT FC131={TOOL_NO 2,BASE_NO 10,IPO_FRAME #BASE,POINT2[] " ",TQ_STATE FALSE}
DECL E6POS XCAux131={X 48.460,Y 116.990,Z -42.760,A 0.000,B 11.750,C -30.130}
DECL E6POS XCDes131={X -48.460,Y 116.990,Z -42.760,A -0.000,B -11.750,C -30.130}
DECL LDAT LCPDATP132={VEL 1,ACC 100,APO_DIST 5,APO_FAC 50.0,ORI_TYP #VAR,CIRC_TYP #BASE,JERK_FAC 50.0}
DECL FDAT FP132={TOOL_NO 2,BASE_NO 10,IPO_FRAME #BASE,POINT2[] " ",TQ_STATE FALSE}
DECL E6POS XP132={X -60.420,Y 111.290,Z -42.760,A -0.000,B -14.700,C -28.900}
DECL LDAT LCPDATP133={VEL 1,ACC 100,APO_DIST 5,APO_FAC 50.0,ORI_TYP #VAR,CIRC_TYP #BASE,JERK_FAC 50.0}
DECL FDAT FP133={TOOL_NO 2,BASE_NO 10,IPO_FRAME #BASE,POINT2[] " ",TQ_STATE FALSE}
DECL E6POS XP133={X -56.530,Y 104.120,Z -36.070,A 0.000,B -20.270,C -42.850}
DECL LDAT LCPDATC134={VEL 0.1,ACC 100,APO_DIST 5,APO_FAC 50.0,ORI_TYP #VAR,CIRC_TYP #BASE,JERK_FAC 50.0}
DECL FDAT FC134={TOOL_NO 2,BASE_NO 10,IPO_FRAME #BASE,POINT2[] " ",TQ_STATE FALSE}
DECL E6POS XCAux134={X -45.340,Y 109.450,Z -36.070,A -0.000,B -16.130,C -44.280}
DECL E6POS XCDes134={X 45.340,Y 109.450,Z -36.070,A -0.000,B 16.130,C -44.280}
DECL LDAT LCPDATP135={VEL 1,ACC 100,APO_DIST 5,APO_FAC 50.0,ORI_TYP #VAR,CIRC_TYP #BASE,JERK_FAC 50.0}
DECL FDAT FP135={TOOL_NO 2,BASE_NO 10,IPO_FRAME #BASE,POINT2[] " ",TQ_STATE FALSE}
DECL E6POS XP135={X 56.530,Y 104.120,Z -36.070,A -0.000,B 20.270,C -42.850}
DECL LDAT LCPDATP136={VEL 0.5,ACC 100,APO_DIST 5,APO_FAC 50.0,ORI_TYP #VAR,CIRC_TYP #BASE,JERK_FAC 50.0}
DECL FDAT FP136={TOOL_NO 2,BASE_NO 10,IPO_FRAME #BASE,POINT2[] " ",TQ_STATE FALSE}
DECL E6POS XP136={X 123.850,Y 136.020,Z 98.320,A 0.000,B 0.000,C 180.000}
DECL LDAT LCPDATP137={VEL 0.5,ACC 100,APO_DIST 5,APO_FAC 50.0,ORI_TYP #VAR,CIRC_TYP #BASE,JERK_FAC 50.0}
DECL FDAT FP137={TOOL_NO 2,BASE_NO 10,IPO_FRAME #BASE,POINT2[] " ",TQ_STATE FALSE}
DECL E6POS XP137={X 123.850,Y 236.020,Z 98.320,A 0.000,B 0.000,C 180.000}
DECL LDAT LCPDATP138={VEL 1.0,ACC 100,APO_DIST 5,APO_FAC 50.0,ORI_TYP #VAR,CIRC_TYP #BASE,JERK_FAC 50.0}
DECL FDAT FP138={TOOL_NO 2,BASE_NO 10,IPO_FRAME #BASE,POINT2[] " ",TQ_STATE FALSE}
DECL E6POS XP138={X 123.850,Y 380.000,Z -20.000,A 0.000,B 0.000,C 0.000}
DECL LDAT LCPDATP139={VEL 1.0,ACC 100,APO_DIST 5,APO_FAC 50.0,ORI_TYP #VAR,CIRC_TYP #BASE,JERK_FAC 50.0}
DECL FDAT FP139={TOOL_NO 2,BASE_NO 10,IPO_FRAME #BASE,POINT2[] " ",TQ_STATE FALSE}
DECL E6POS XP139={X -58.570,Y 380.000,Z -20.000,A 0.000,B 0.000,C 0.000}
;ENDDAT for Routine_0

ENDDAT
